% RSLogix 500 project DMINFEED - ONSITE - 17-01-07 - AFTER CHANGES.RSS, saved by version 7.00.00.19 %
PROJECT "DMINFEED"    % processor: SLC 500, 1747-L541 %

PROGRAM FILES
  LAD 2 "MAIN"  16 rungs
  LAD 3 "DECK1 TILT"  21 rungs
  LAD 4 "DECK2 TILT"  18 rungs
  LAD 5 "LUGLOADER"  18 rungs
  LAD 6 "SPARE"  1 rungs
  LAD 7 "DECK1 MOTS"  53 rungs
  LAD 8 "EXTRACTFAN"  7 rungs
  LAD 9 "BLOCKTX"  2 rungs
  LAD 14 "DECK2 MOTS"  23 rungs
  LAD 15 "ENCODER"  4 rungs
  LAD 16 "FEED_CONTR"  7 rungs
  LAD 17 "SCELUGLOAD"  11 rungs
  LAD 18 "REPORTING"  4 rungs
  LAD 20 "FILLET SYS"  28 rungs

DATA FILES
  O0 OUTPUT  39 elements
  I1 INPUT  46 elements
  S2 STATUS  164 elements
  B3 BINARY  100 elements
  T4 TIMER  100 elements
  C5 COUNTER  100 elements
  R6 CONTROL  1 elements
  N7 INTEGER  100 elements
  F8 FLOAT  1 elements
  N9 REMOTE IO  20 elements
  N10   100 elements
  N11 SCE SYSTEM  101 elements
  T12 SCE TIMER  11 elements
  N13   42 elements
  T14   30 elements
  C15   30 elements
  B16   100 elements

LADDER 2 "MAIN"
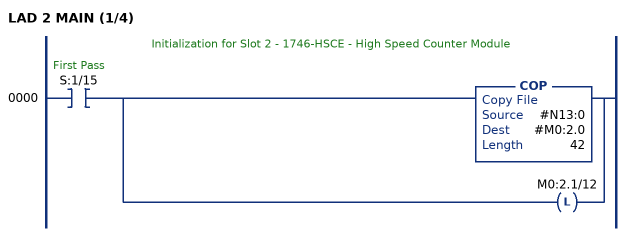
% Rung: 0 %
% Initialization for Slot 2 - 1746-HSCE - High Speed Counter Module %
SOR XIC S:1/15 BST COP #N13:0 #M0:2.0 42 NXB OTL M0:2.1/12 BND EOR
%   S:1/15  "First Pass" %

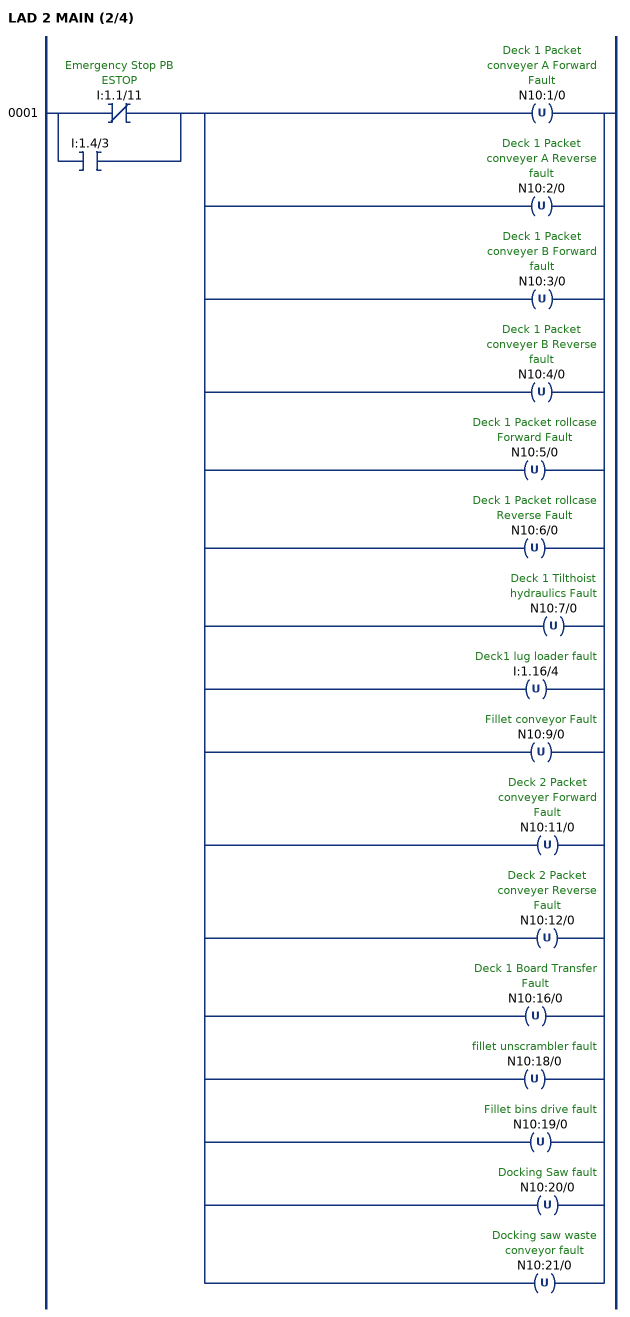
% Rung: 1 %
SOR BST XIO I:1.1/11 NXB XIC I:1.4/3 BND BST OTU N10:1/0 NXB OTU N10:2/0 NXB OTU N10:3/0 NXB OTU N10:4/0 NXB OTU N10:5/0 NXB OTU N10:6/0 NXB OTU N10:7/0 NXB OTU I:1.16/4 NXB OTU N10:9/0 NXB OTU N10:11/0 NXB OTU N10:12/0 NXB OTU N10:16/0 NXB OTU N10:18/0 NXB OTU N10:19/0 NXB OTU N10:20/0 NXB OTU N10:21/0 BND EOR
%   I:1.1/11  ESTOP  "Emergency Stop PB" %
%   N10:1/0  "Deck 1 Packet conveyer A Forward Fault" %
%   N10:2/0  "Deck 1 Packet conveyer A Reverse fault" %
%   N10:3/0  "Deck 1 Packet conveyer B Forward fault" %
%   N10:4/0  "Deck 1 Packet conveyer B Reverse fault" %
%   N10:5/0  "Deck 1 Packet rollcase Forward Fault" %
%   N10:6/0  "Deck 1 Packet rollcase Reverse Fault" %
%   N10:7/0  "Deck 1 Tilthoist hydraulics Fault" %
%   I:1.16/4  "Deck1 lug loader fault" %
%   N10:9/0  "Fillet conveyor Fault" %
%   N10:11/0  "Deck 2 Packet conveyer Forward Fault" %
%   N10:12/0  "Deck 2 Packet conveyer Reverse Fault" %
%   N10:16/0  "Deck 1 Board Transfer Fault" %
%   N10:18/0  "fillet unscrambler fault" %
%   N10:19/0  "Fillet bins drive fault" %
%   N10:20/0  "Docking Saw fault" %
%   N10:21/0  "Docking saw waste conveyor fault" %

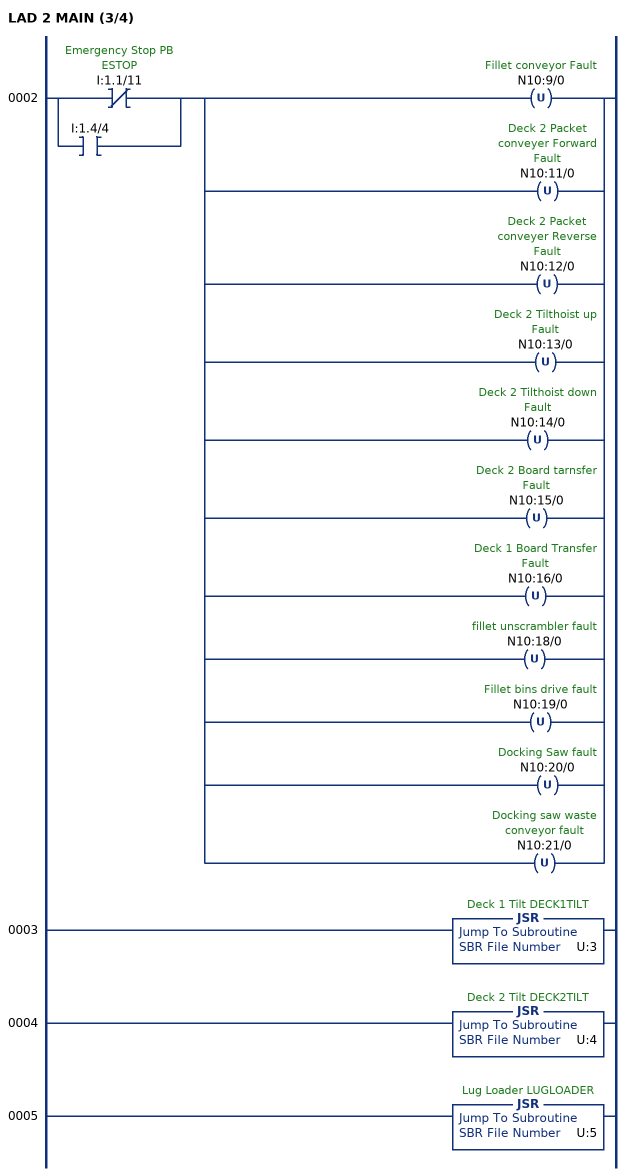
% Rung: 2 %
SOR BST XIO I:1.1/11 NXB XIC I:1.4/4 BND BST OTU N10:9/0 NXB OTU N10:11/0 NXB OTU N10:12/0 NXB OTU N10:13/0 NXB OTU N10:14/0 NXB OTU N10:15/0 NXB OTU N10:16/0 NXB OTU N10:18/0 NXB OTU N10:19/0 NXB OTU N10:20/0 NXB OTU N10:21/0 BND EOR
%   I:1.1/11  ESTOP  "Emergency Stop PB" %
%   N10:9/0  "Fillet conveyor Fault" %
%   N10:11/0  "Deck 2 Packet conveyer Forward Fault" %
%   N10:12/0  "Deck 2 Packet conveyer Reverse Fault" %
%   N10:13/0  "Deck 2 Tilthoist up Fault" %
%   N10:14/0  "Deck 2 Tilthoist down Fault" %
%   N10:15/0  "Deck 2 Board tarnsfer Fault" %
%   N10:16/0  "Deck 1 Board Transfer Fault" %
%   N10:18/0  "fillet unscrambler fault" %
%   N10:19/0  "Fillet bins drive fault" %
%   N10:20/0  "Docking Saw fault" %
%   N10:21/0  "Docking saw waste conveyor fault" %
% Rung: 3 %
SOR JSR U:3 EOR
%   U:3  DECK1TILT  "Deck 1 Tilt" %
% Rung: 4 %
SOR JSR U:4 EOR
%   U:4  DECK2TILT  "Deck 2 Tilt" %
% Rung: 5 %
SOR JSR U:5 EOR
%   U:5  LUGLOADER  "Lug Loader" %

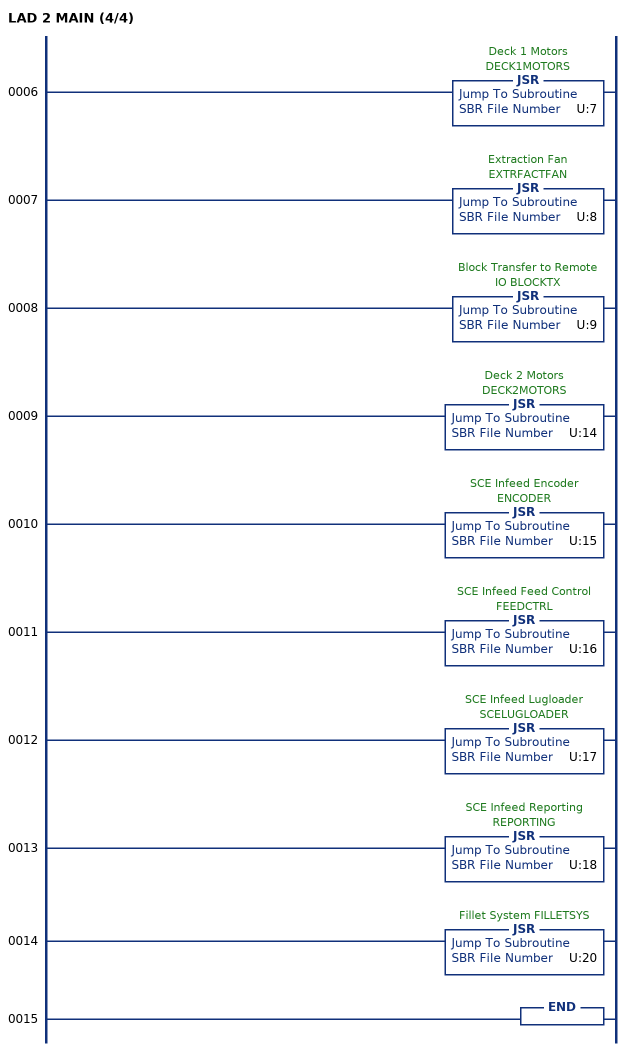
% Rung: 6 %
SOR JSR U:7 EOR
%   U:7  DECK1MOTORS  "Deck 1 Motors" %
% Rung: 7 %
SOR JSR U:8 EOR
%   U:8  EXTRFACTFAN  "Extraction Fan" %
% Rung: 8 %
SOR JSR U:9 EOR
%   U:9  BLOCKTX  "Block Transfer to Remote IO" %
% Rung: 9 %
SOR JSR U:14 EOR
%   U:14  DECK2MOTORS  "Deck 2 Motors" %
% Rung: 10 %
SOR JSR U:15 EOR
%   U:15  ENCODER  "SCE Infeed Encoder" %
% Rung: 11 %
SOR JSR U:16 EOR
%   U:16  FEEDCTRL  "SCE Infeed Feed Control" %
% Rung: 12 %
SOR JSR U:17 EOR
%   U:17  SCELUGLOADER  "SCE Infeed Lugloader" %
% Rung: 13 %
SOR JSR U:18 EOR
%   U:18  REPORTING  "SCE Infeed Reporting" %
% Rung: 14 %
SOR JSR U:20 EOR
%   U:20  FILLETSYS  "Fillet System" %
% Rung: 15 %
SOR END EOR

LADDER 3 "DECK1 TILT"
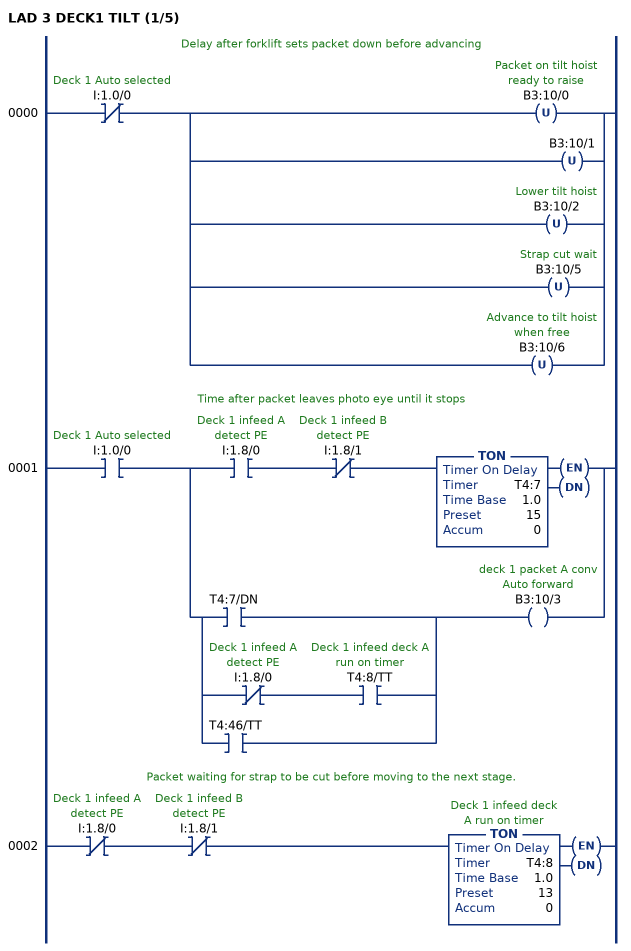
% Rung: 0 %
% Delay after forklift sets packet down before advancing %
SOR XIO I:1.0/0 BST OTU B3:10/0 NXB OTU B3:10/1 NXB OTU B3:10/2 NXB OTU B3:10/5 NXB OTU B3:10/6 BND EOR
%   I:1.0/0  "Deck 1 Auto selected" %
%   B3:10/0  "Packet on tilt hoist ready to raise" %
%   B3:10/2  "Lower tilt hoist" %
%   B3:10/5  "Strap cut wait" %
%   B3:10/6  "Advance to tilt hoist when free" %
% Rung: 1 %
% Time after packet leaves photo eye until it stops %
SOR XIC I:1.0/0 BST XIC I:1.8/0 XIO I:1.8/1 TON T4:7 1.0 15 0 NXB BST XIC T4:7/DN NXB XIO I:1.8/0 XIC T4:8/TT NXB XIC T4:46/TT BND OTE B3:10/3 BND EOR
%   I:1.0/0  "Deck 1 Auto selected" %
%   I:1.8/0  "Deck 1 infeed A detect PE" %
%   I:1.8/1  "Deck 1 infeed B detect PE" %
%   T4:8  "Deck 1 infeed deck A run on timer" %
%   B3:10/3  "deck 1 packet A conv Auto forward" %
% Rung: 2 %
% Packet waiting for strap to be cut before moving to the next stage. %
SOR XIO I:1.8/0 XIO I:1.8/1 TON T4:8 1.0 13 0 EOR
%   I:1.8/0  "Deck 1 infeed A detect PE" %
%   I:1.8/1  "Deck 1 infeed B detect PE" %
%   T4:8  "Deck 1 infeed deck A run on timer" %

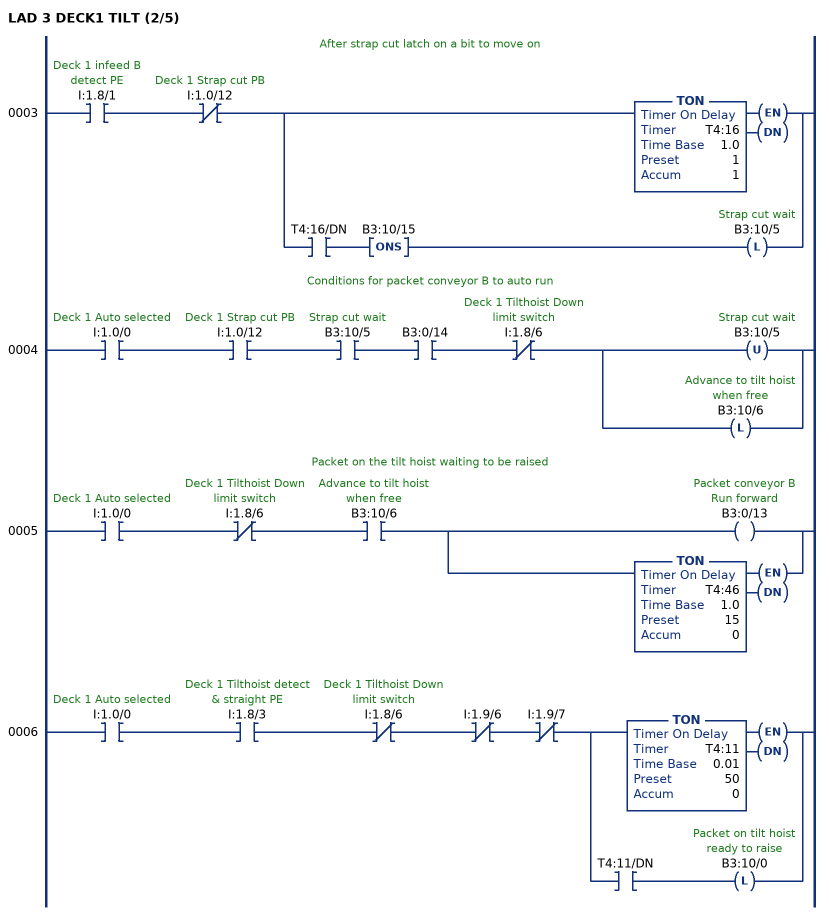
% Rung: 3 %
% After strap cut latch on a bit to move on %
SOR XIC I:1.8/1 XIO I:1.0/12 BST TON T4:16 1.0 1 1 NXB XIC T4:16/DN OSR B3:10/15 OTL B3:10/5 BND EOR
%   I:1.8/1  "Deck 1 infeed B detect PE" %
%   I:1.0/12  "Deck 1 Strap cut PB" %
%   B3:10/5  "Strap cut wait" %
% Rung: 4 %
% Conditions for packet conveyor B to auto run %
SOR XIC I:1.0/0 XIC I:1.0/12 XIC B3:10/5 XIC B3:0/14 XIO I:1.8/6 BST OTU B3:10/5 NXB OTL B3:10/6 BND EOR
%   I:1.0/0  "Deck 1 Auto selected" %
%   I:1.0/12  "Deck 1 Strap cut PB" %
%   B3:10/5  "Strap cut wait" %
%   I:1.8/6  "Deck 1 Tilthoist Down limit switch" %
%   B3:10/6  "Advance to tilt hoist when free" %
% Rung: 5 %
% Packet on the tilt hoist waiting to be raised %
SOR XIC I:1.0/0 XIO I:1.8/6 XIC B3:10/6 BST OTE B3:0/13 NXB TON T4:46 1.0 15 0 BND EOR
%   I:1.0/0  "Deck 1 Auto selected" %
%   I:1.8/6  "Deck 1 Tilthoist Down limit switch" %
%   B3:10/6  "Advance to tilt hoist when free" %
%   B3:0/13  "Packet conveyor B Run forward" %
% Rung: 6 %
SOR XIC I:1.0/0 XIC I:1.8/3 XIO I:1.8/6 XIO I:1.9/6 XIO I:1.9/7 BST TON T4:11 0.01 50 0 NXB XIC T4:11/DN OTL B3:10/0 BND EOR
%   I:1.0/0  "Deck 1 Auto selected" %
%   I:1.8/3  "Deck 1 Tilthoist detect & straight PE" %
%   I:1.8/6  "Deck 1 Tilthoist Down limit switch" %
%   B3:10/0  "Packet on tilt hoist ready to raise" %

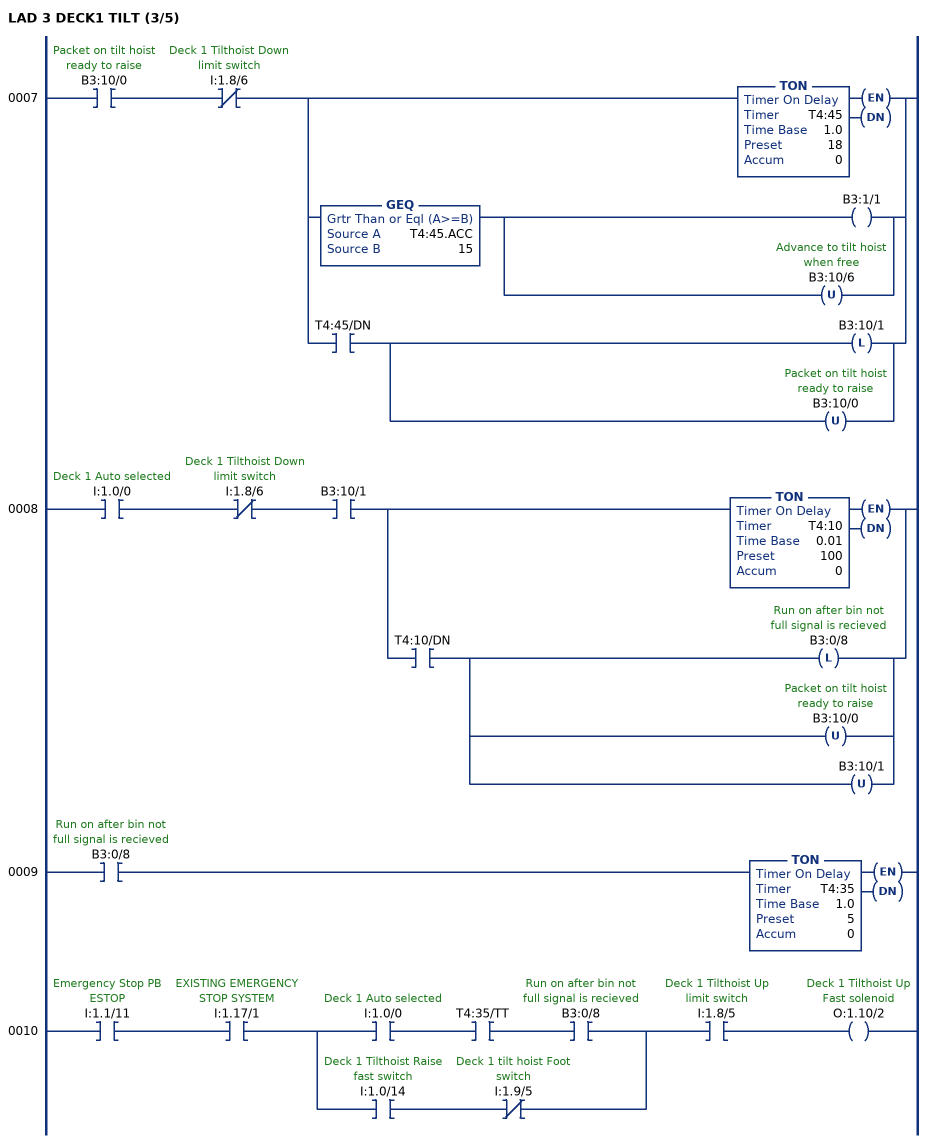
% Rung: 7 %
SOR XIC B3:10/0 XIO I:1.8/6 BST TON T4:45 1.0 18 0 NXB GEQ T4:45.ACC 15 BST OTE B3:1/1 NXB OTU B3:10/6 BND NXB XIC T4:45/DN BST OTL B3:10/1 NXB OTU B3:10/0 BND BND EOR
%   B3:10/0  "Packet on tilt hoist ready to raise" %
%   I:1.8/6  "Deck 1 Tilthoist Down limit switch" %
%   B3:10/6  "Advance to tilt hoist when free" %
% Rung: 8 %
SOR XIC I:1.0/0 XIO I:1.8/6 XIC B3:10/1 BST TON T4:10 0.01 100 0 NXB XIC T4:10/DN BST OTL B3:0/8 NXB OTU B3:10/0 NXB OTU B3:10/1 BND BND EOR
%   I:1.0/0  "Deck 1 Auto selected" %
%   I:1.8/6  "Deck 1 Tilthoist Down limit switch" %
%   B3:0/8  "Run on after bin not full signal is recieved" %
%   B3:10/0  "Packet on tilt hoist ready to raise" %
% Rung: 9 %
SOR XIC B3:0/8 TON T4:35 1.0 5 0 EOR
%   B3:0/8  "Run on after bin not full signal is recieved" %
% Rung: 10 %
SOR XIC I:1.1/11 XIC I:1.17/1 BST XIC I:1.0/0 XIC T4:35/TT XIC B3:0/8 NXB XIC I:1.0/14 XIO I:1.9/5 BND XIC I:1.8/5 OTE O:1.10/2 EOR
%   I:1.1/11  ESTOP  "Emergency Stop PB" %
%   I:1.17/1  "EXISTING EMERGENCY STOP SYSTEM" %
%   I:1.0/0  "Deck 1 Auto selected" %
%   B3:0/8  "Run on after bin not full signal is recieved" %
%   I:1.0/14  "Deck 1 Tilthoist Raise fast switch" %
%   I:1.9/5  "Deck 1 tilt hoist Foot switch" %
%   I:1.8/5  "Deck 1 Tilthoist Up limit switch" %
%   O:1.10/2  "Deck 1 Tilthoist Up Fast solenoid" %

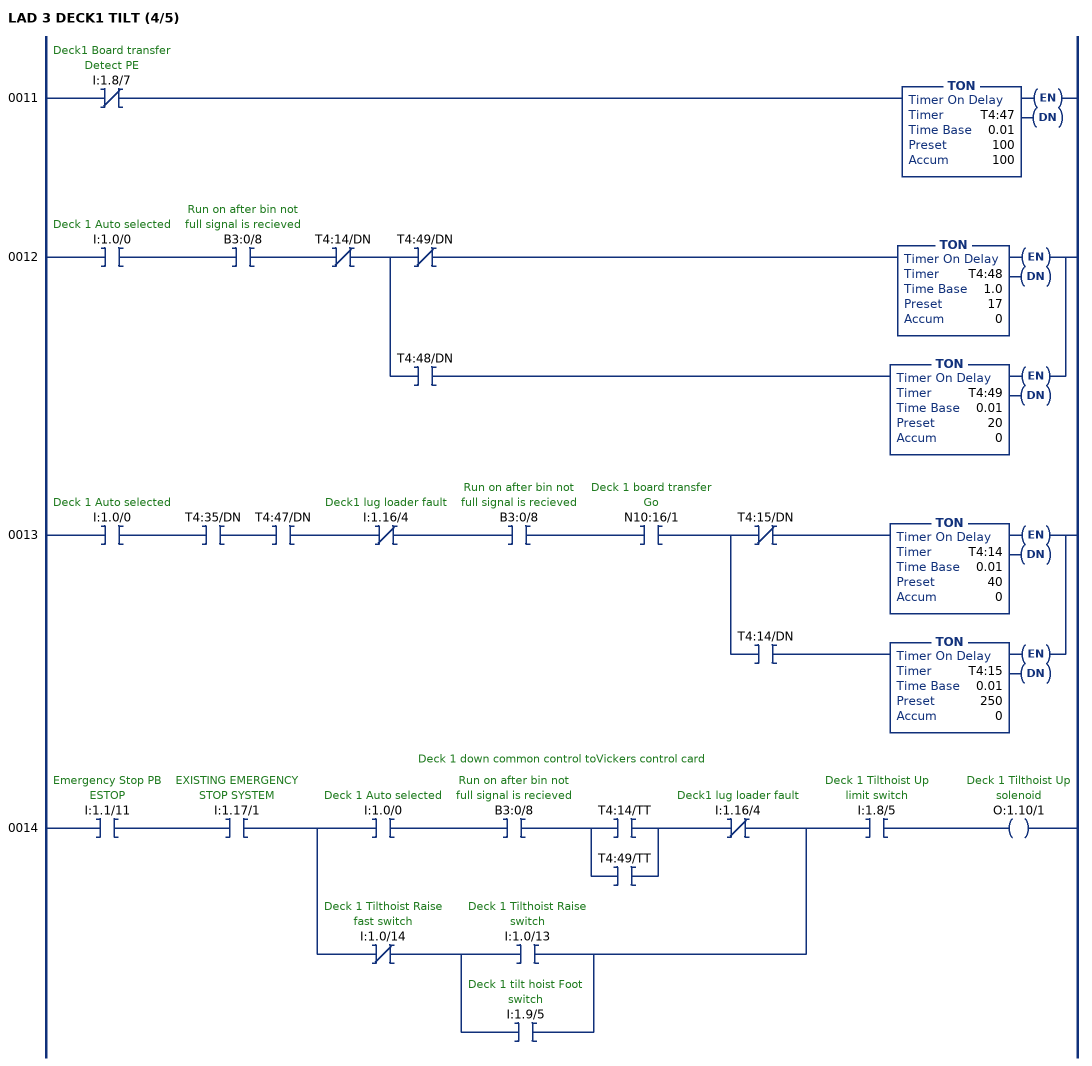
% Rung: 11 %
SOR XIO I:1.8/7 TON T4:47 0.01 100 100 EOR
%   I:1.8/7  "Deck1 Board transfer Detect PE" %
% Rung: 12 %
SOR XIC I:1.0/0 XIC B3:0/8 XIO T4:14/DN BST XIO T4:49/DN TON T4:48 1.0 17 0 NXB XIC T4:48/DN TON T4:49 0.01 20 0 BND EOR
%   I:1.0/0  "Deck 1 Auto selected" %
%   B3:0/8  "Run on after bin not full signal is recieved" %
% Rung: 13 %
SOR XIC I:1.0/0 XIC T4:35/DN XIC T4:47/DN XIO I:1.16/4 XIC B3:0/8 XIC N10:16/1 BST XIO T4:15/DN TON T4:14 0.01 40 0 NXB XIC T4:14/DN TON T4:15 0.01 250 0 BND EOR
%   I:1.0/0  "Deck 1 Auto selected" %
%   I:1.16/4  "Deck1 lug loader fault" %
%   B3:0/8  "Run on after bin not full signal is recieved" %
%   N10:16/1  "Deck 1 board transfer Go" %
% Rung: 14 %
% Deck 1 down common control toVickers control card %
SOR XIC I:1.1/11 XIC I:1.17/1 BST XIC I:1.0/0 XIC B3:0/8 BST XIC T4:14/TT NXB XIC T4:49/TT BND XIO I:1.16/4 NXB XIO I:1.0/14 BST XIC I:1.0/13 NXB XIC I:1.9/5 BND BND XIC I:1.8/5 OTE O:1.10/1 EOR
%   I:1.1/11  ESTOP  "Emergency Stop PB" %
%   I:1.17/1  "EXISTING EMERGENCY STOP SYSTEM" %
%   I:1.0/0  "Deck 1 Auto selected" %
%   B3:0/8  "Run on after bin not full signal is recieved" %
%   I:1.16/4  "Deck1 lug loader fault" %
%   I:1.0/14  "Deck 1 Tilthoist Raise fast switch" %
%   I:1.0/13  "Deck 1 Tilthoist Raise switch" %
%   I:1.9/5  "Deck 1 tilt hoist Foot switch" %
%   I:1.8/5  "Deck 1 Tilthoist Up limit switch" %
%   O:1.10/1  "Deck 1 Tilthoist Up solenoid" %

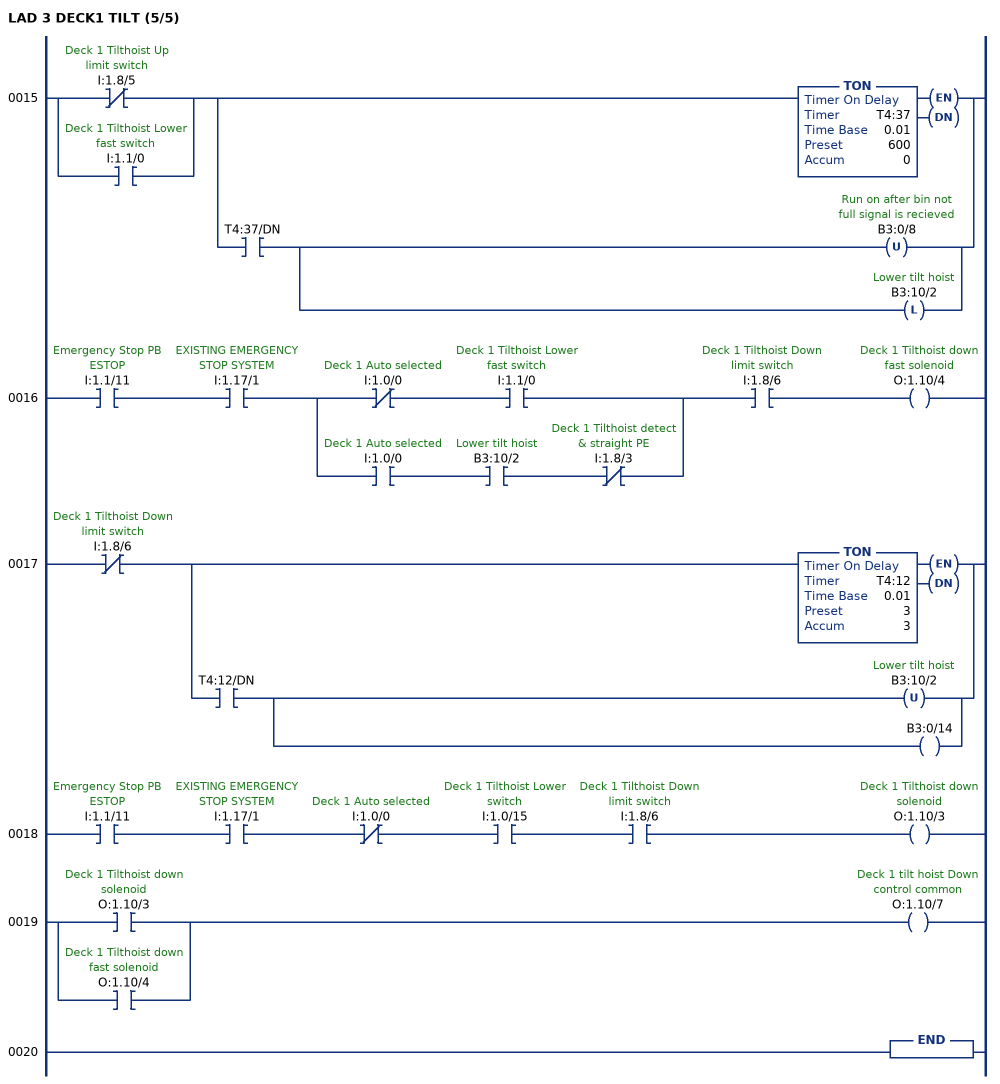
% Rung: 15 %
SOR BST XIO I:1.8/5 NXB XIC I:1.1/0 BND BST TON T4:37 0.01 600 0 NXB XIC T4:37/DN BST OTU B3:0/8 NXB OTL B3:10/2 BND BND EOR
%   I:1.8/5  "Deck 1 Tilthoist Up limit switch" %
%   I:1.1/0  "Deck 1 Tilthoist Lower fast switch" %
%   B3:0/8  "Run on after bin not full signal is recieved" %
%   B3:10/2  "Lower tilt hoist" %
% Rung: 16 %
SOR XIC I:1.1/11 XIC I:1.17/1 BST XIO I:1.0/0 XIC I:1.1/0 NXB XIC I:1.0/0 XIC B3:10/2 XIO I:1.8/3 BND XIC I:1.8/6 OTE O:1.10/4 EOR
%   I:1.1/11  ESTOP  "Emergency Stop PB" %
%   I:1.17/1  "EXISTING EMERGENCY STOP SYSTEM" %
%   I:1.0/0  "Deck 1 Auto selected" %
%   I:1.1/0  "Deck 1 Tilthoist Lower fast switch" %
%   B3:10/2  "Lower tilt hoist" %
%   I:1.8/3  "Deck 1 Tilthoist detect & straight PE" %
%   I:1.8/6  "Deck 1 Tilthoist Down limit switch" %
%   O:1.10/4  "Deck 1 Tilthoist down fast solenoid" %
% Rung: 17 %
SOR XIO I:1.8/6 BST TON T4:12 0.01 3 3 NXB XIC T4:12/DN BST OTU B3:10/2 NXB OTE B3:0/14 BND BND EOR
%   I:1.8/6  "Deck 1 Tilthoist Down limit switch" %
%   B3:10/2  "Lower tilt hoist" %
% Rung: 18 %
SOR XIC I:1.1/11 XIC I:1.17/1 XIO I:1.0/0 XIC I:1.0/15 XIC I:1.8/6 OTE O:1.10/3 EOR
%   I:1.1/11  ESTOP  "Emergency Stop PB" %
%   I:1.17/1  "EXISTING EMERGENCY STOP SYSTEM" %
%   I:1.0/0  "Deck 1 Auto selected" %
%   I:1.0/15  "Deck 1 Tilthoist Lower switch" %
%   I:1.8/6  "Deck 1 Tilthoist Down limit switch" %
%   O:1.10/3  "Deck 1 Tilthoist down solenoid" %
% Rung: 19 %
SOR BST XIC O:1.10/3 NXB XIC O:1.10/4 BND OTE O:1.10/7 EOR
%   O:1.10/3  "Deck 1 Tilthoist down solenoid" %
%   O:1.10/4  "Deck 1 Tilthoist down fast solenoid" %
%   O:1.10/7  "Deck 1 tilt hoist Down control common" %
% Rung: 20 %
SOR END EOR

LADDER 4 "DECK2 TILT"
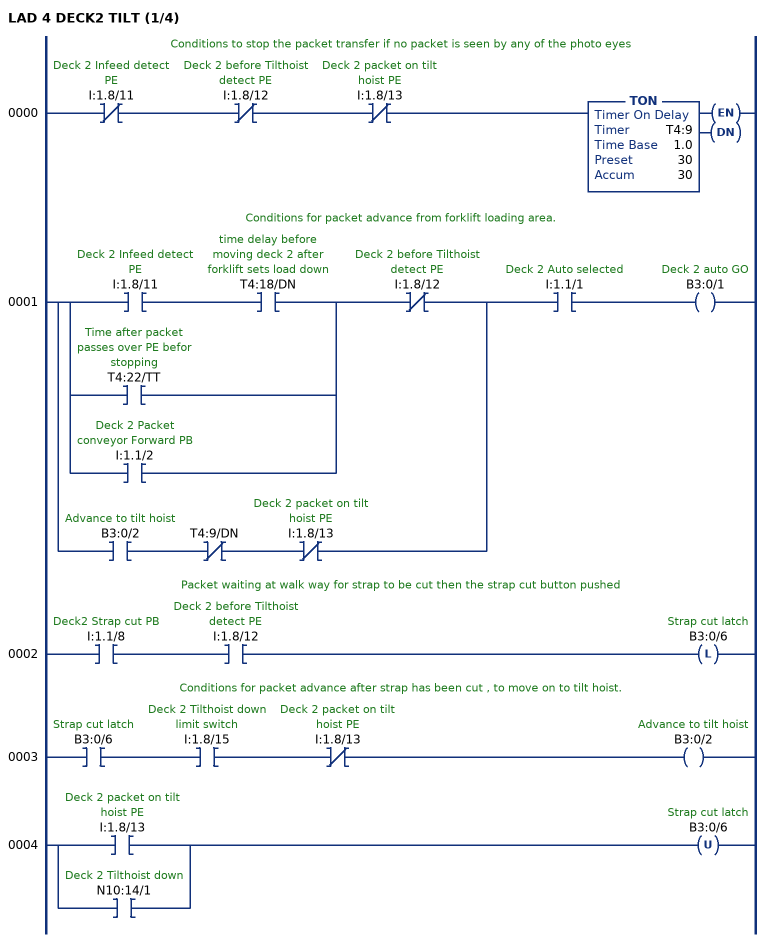
% Rung: 0 %
% Conditions to stop the packet transfer if no packet is seen by any of the photo eyes %
SOR XIO I:1.8/11 XIO I:1.8/12 XIO I:1.8/13 TON T4:9 1.0 30 30 EOR
%   I:1.8/11  "Deck 2 Infeed detect PE" %
%   I:1.8/12  "Deck 2 before Tilthoist detect PE" %
%   I:1.8/13  "Deck 2 packet on tilt hoist PE" %
% Rung: 1 %
% Conditions for packet advance from forklift loading area. %
SOR BST BST XIC I:1.8/11 XIC T4:18/DN NXB BST XIC T4:22/TT NXB XIC I:1.1/2 BND BND XIO I:1.8/12 NXB XIC B3:0/2 XIO T4:9/DN XIO I:1.8/13 BND XIC I:1.1/1 OTE B3:0/1 EOR
%   I:1.8/11  "Deck 2 Infeed detect PE" %
%   T4:18  "time delay before moving deck 2 after forklift sets load down" %
%   T4:22  "Time after packet passes over PE befor stopping" %
%   I:1.1/2  "Deck 2 Packet conveyor Forward PB" %
%   I:1.8/12  "Deck 2 before Tilthoist detect PE" %
%   B3:0/2  "Advance to tilt hoist" %
%   I:1.8/13  "Deck 2 packet on tilt hoist PE" %
%   I:1.1/1  "Deck 2 Auto selected" %
%   B3:0/1  "Deck 2 auto GO" %
% Rung: 2 %
% Packet waiting at walk way for strap to be cut then the strap cut button pushed %
SOR XIC I:1.1/8 XIC I:1.8/12 OTL B3:0/6 EOR
%   I:1.1/8  "Deck2 Strap cut PB" %
%   I:1.8/12  "Deck 2 before Tilthoist detect PE" %
%   B3:0/6  "Strap cut latch" %
% Rung: 3 %
% Conditions for packet advance after strap has been cut , to move on to tilt hoist. %
SOR XIC B3:0/6 XIC I:1.8/15 XIO I:1.8/13 OTE B3:0/2 EOR
%   B3:0/6  "Strap cut latch" %
%   I:1.8/15  "Deck 2 Tilthoist down limit switch" %
%   I:1.8/13  "Deck 2 packet on tilt hoist PE" %
%   B3:0/2  "Advance to tilt hoist" %
% Rung: 4 %
SOR BST XIC I:1.8/13 NXB XIC N10:14/1 BND OTU B3:0/6 EOR
%   I:1.8/13  "Deck 2 packet on tilt hoist PE" %
%   N10:14/1  "Deck 2 Tilthoist down" %
%   B3:0/6  "Strap cut latch" %

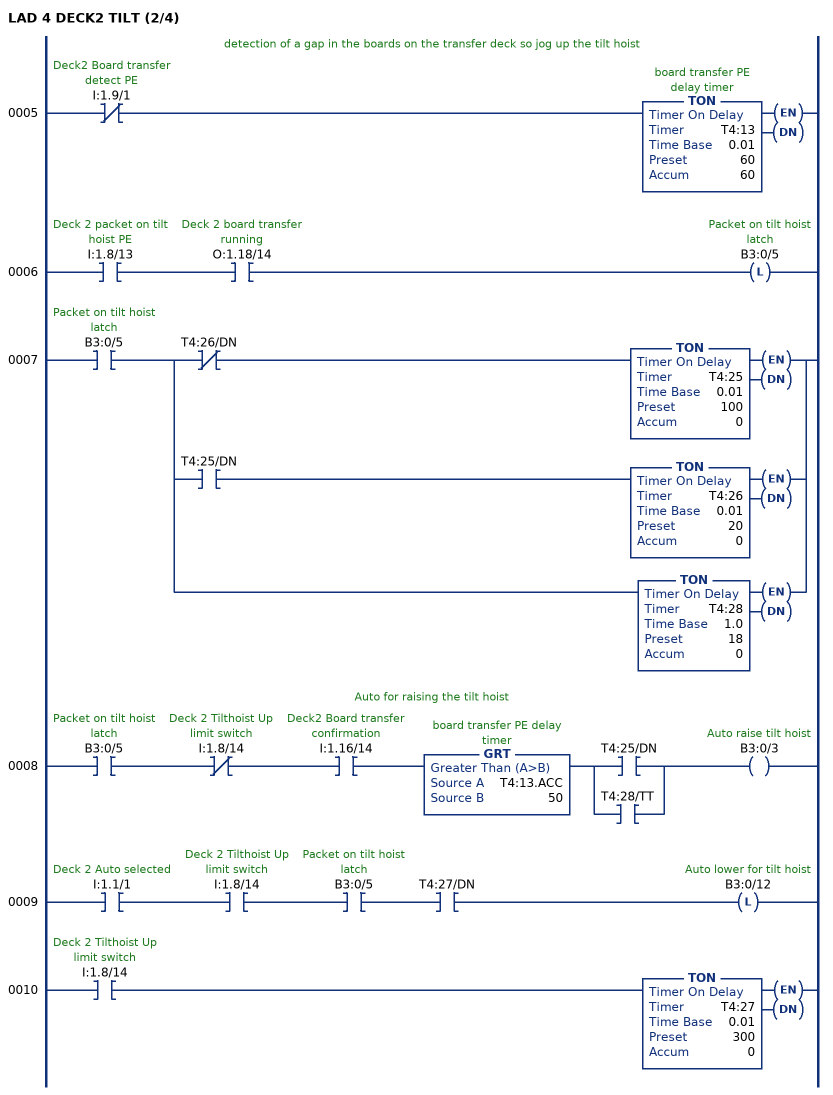
% Rung: 5 %
% detection of a gap in the boards on the transfer deck so jog up the tilt hoist %
SOR XIO I:1.9/1 TON T4:13 0.01 60 60 EOR
%   I:1.9/1  "Deck2 Board transfer detect PE" %
%   T4:13  "board transfer PE delay timer" %
% Rung: 6 %
SOR XIC I:1.8/13 XIC O:1.18/14 OTL B3:0/5 EOR
%   I:1.8/13  "Deck 2 packet on tilt hoist PE" %
%   O:1.18/14  "Deck 2 board transfer running" %
%   B3:0/5  "Packet on tilt hoist latch" %
% Rung: 7 %
SOR XIC B3:0/5 BST XIO T4:26/DN TON T4:25 0.01 100 0 NXB BST XIC T4:25/DN TON T4:26 0.01 20 0 NXB TON T4:28 1.0 18 0 BND BND EOR
%   B3:0/5  "Packet on tilt hoist latch" %
% Rung: 8 %
% Auto for raising the tilt hoist %
SOR XIC B3:0/5 XIO I:1.8/14 XIC I:1.16/14 GRT T4:13.ACC 50 BST XIC T4:25/DN NXB XIC T4:28/TT BND OTE B3:0/3 EOR
%   B3:0/5  "Packet on tilt hoist latch" %
%   I:1.8/14  "Deck 2 Tilthoist Up limit switch" %
%   I:1.16/14  "Deck2 Board transfer confirmation" %
%   T4:13  "board transfer PE delay timer" %
%   B3:0/3  "Auto raise tilt hoist" %
% Rung: 9 %
SOR XIC I:1.1/1 XIC I:1.8/14 XIC B3:0/5 XIC T4:27/DN OTL B3:0/12 EOR
%   I:1.1/1  "Deck 2 Auto selected" %
%   I:1.8/14  "Deck 2 Tilthoist Up limit switch" %
%   B3:0/5  "Packet on tilt hoist latch" %
%   B3:0/12  "Auto lower for tilt hoist" %
% Rung: 10 %
SOR XIC I:1.8/14 TON T4:27 0.01 300 0 EOR
%   I:1.8/14  "Deck 2 Tilthoist Up limit switch" %

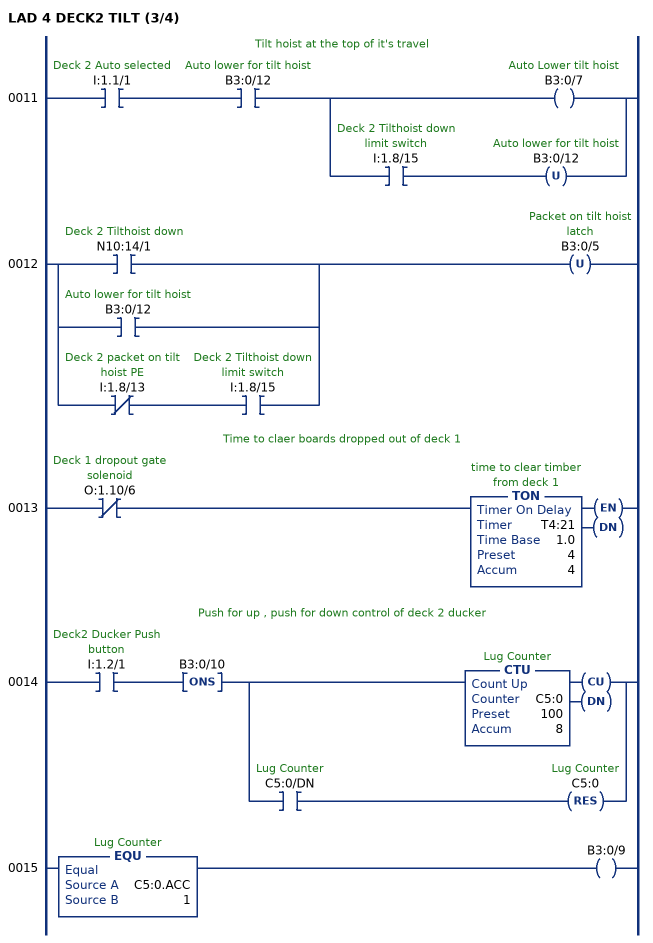
% Rung: 11 %
% Tilt hoist at the top of it's travel %
SOR XIC I:1.1/1 XIC B3:0/12 BST OTE B3:0/7 NXB XIC I:1.8/15 OTU B3:0/12 BND EOR
%   I:1.1/1  "Deck 2 Auto selected" %
%   B3:0/12  "Auto lower for tilt hoist" %
%   B3:0/7  "Auto Lower tilt hoist" %
%   I:1.8/15  "Deck 2 Tilthoist down limit switch" %
% Rung: 12 %
SOR BST BST XIC N10:14/1 NXB XIC B3:0/12 BND NXB XIO I:1.8/13 XIC I:1.8/15 BND OTU B3:0/5 EOR
%   N10:14/1  "Deck 2 Tilthoist down" %
%   B3:0/12  "Auto lower for tilt hoist" %
%   I:1.8/13  "Deck 2 packet on tilt hoist PE" %
%   I:1.8/15  "Deck 2 Tilthoist down limit switch" %
%   B3:0/5  "Packet on tilt hoist latch" %
% Rung: 13 %
% Time to claer boards dropped out of deck 1 %
SOR XIO O:1.10/6 TON T4:21 1.0 4 4 EOR
%   O:1.10/6  "Deck 1 dropout gate solenoid" %
%   T4:21  "time to clear timber from deck 1" %
% Rung: 14 %
% Push for up , push for down control of deck 2 ducker %
SOR XIC I:1.2/1 OSR B3:0/10 BST CTU C5:0 100 8 NXB XIC C5:0/DN RES C5:0 BND EOR
%   I:1.2/1  "Deck2 Ducker Push button" %
%   C5:0  "Lug Counter" %
% Rung: 15 %
SOR EQU C5:0.ACC 1 OTE B3:0/9 EOR
%   C5:0  "Lug Counter" %

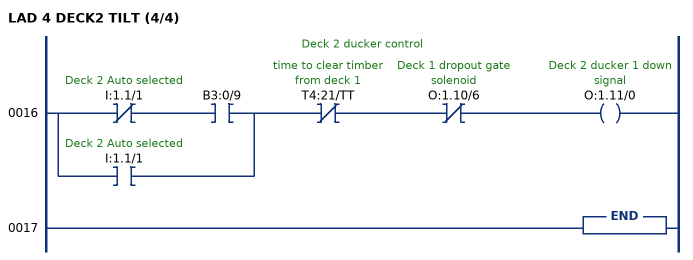
% Rung: 16 %
% Deck 2 ducker control %
SOR BST XIO I:1.1/1 XIC B3:0/9 NXB XIC I:1.1/1 BND XIO T4:21/TT XIO O:1.10/6 OTE O:1.11/0 EOR
%   I:1.1/1  "Deck 2 Auto selected" %
%   T4:21  "time to clear timber from deck 1" %
%   O:1.10/6  "Deck 1 dropout gate solenoid" %
%   O:1.11/0  "Deck 2 ducker 1 down signal" %
% Rung: 17 %
SOR END EOR

LADDER 5 "LUGLOADER"
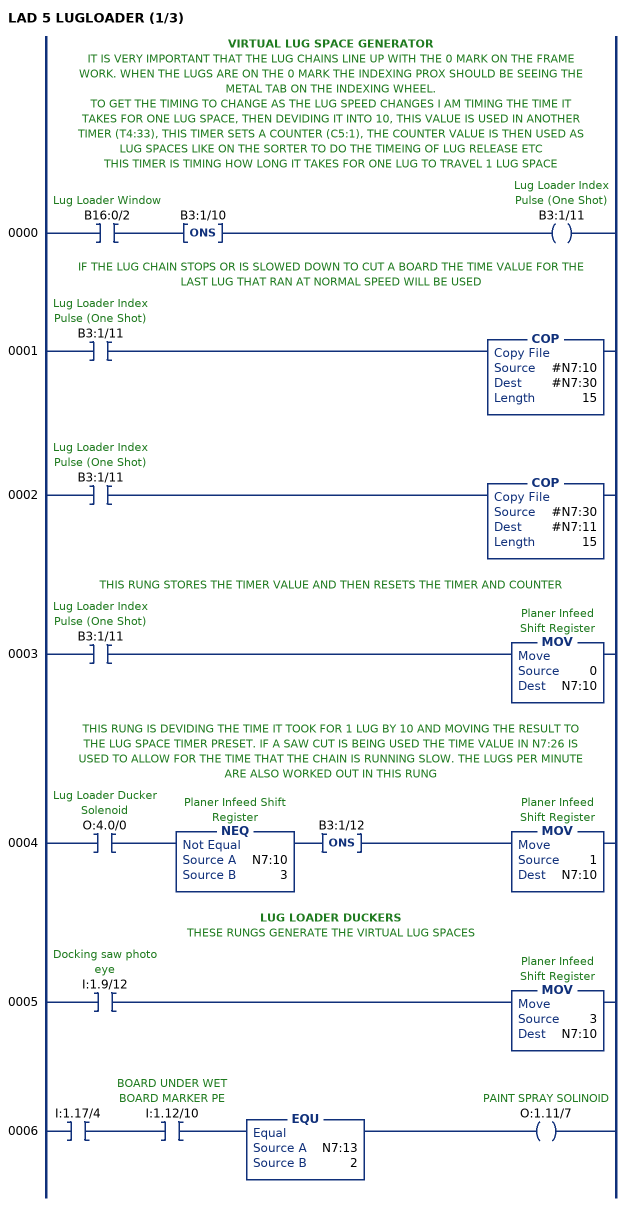
% Rung: 0 %
% TITLE: VIRTUAL LUG SPACE GENERATOR %
% IT IS VERY IMPORTANT THAT THE LUG CHAINS LINE UP WITH THE 0 MARK ON THE FRAME WORK. WHEN THE LUGS ARE ON THE 0 MARK THE INDEXING PROX SHOULD BE SEEING THE METAL TAB ON THE INDEXING WHEEL.
% TO GET THE TIMING TO CHANGE AS THE LUG SPEED CHANGES I AM TIMING THE TIME IT TAKES FOR ONE LUG SPACE, THEN DEVIDING IT INTO 10, THIS VALUE IS USED IN ANOTHER TIMER (T4:33), THIS TIMER SETS A COUNTER (C5:1), THE COUNTER VALUE IS THEN USED AS LUG SPACES LIKE ON THE SORTER TO DO THE TIMEING OF LUG RELEASE ETC
% THIS TIMER IS TIMING HOW LONG IT TAKES FOR ONE LUG TO TRAVEL 1 LUG SPACE %
SOR XIC B16:0/2 OSR B3:1/10 OTE B3:1/11 EOR
%   B16:0/2  "Lug Loader Window" %
%   B3:1/11  "Lug Loader Index Pulse (One Shot)" %
% Rung: 1 %
% IF THE LUG CHAIN STOPS OR IS SLOWED DOWN TO CUT A BOARD THE TIME VALUE FOR THE LAST LUG THAT RAN AT NORMAL SPEED WILL BE USED %
SOR XIC B3:1/11 COP #N7:10 #N7:30 15 EOR
%   B3:1/11  "Lug Loader Index Pulse (One Shot)" %
%   N7:10  "Planer Infeed Shift Register" %
% Rung: 2 %
SOR XIC B3:1/11 COP #N7:30 #N7:11 15 EOR
%   B3:1/11  "Lug Loader Index Pulse (One Shot)" %
% Rung: 3 %
% THIS RUNG STORES THE TIMER VALUE AND THEN RESETS THE TIMER AND COUNTER %
SOR XIC B3:1/11 MOV 0 N7:10 EOR
%   B3:1/11  "Lug Loader Index Pulse (One Shot)" %
%   N7:10  "Planer Infeed Shift Register" %
% Rung: 4 %
% THIS RUNG IS DEVIDING THE TIME IT TOOK FOR 1 LUG BY 10 AND MOVING THE RESULT TO THE LUG SPACE TIMER PRESET. IF A SAW CUT IS BEING USED THE TIME VALUE IN N7:26 IS USED TO ALLOW FOR THE TIME THAT THE CHAIN IS RUNNING SLOW. THE LUGS PER MINUTE ARE ALSO WORKED OUT IN THIS RUNG %
SOR XIC O:4.0/0 NEQ N7:10 3 OSR B3:1/12 MOV 1 N7:10 EOR
%   O:4.0/0  "Lug Loader Ducker Solenoid" %
%   N7:10  "Planer Infeed Shift Register" %
% Rung: 5 %
% TITLE: LUG LOADER DUCKERS %
% THESE RUNGS GENERATE THE VIRTUAL LUG SPACES %
SOR XIC I:1.9/12 MOV 3 N7:10 EOR
%   I:1.9/12  "Docking saw photo eye" %
%   N7:10  "Planer Infeed Shift Register" %
% Rung: 6 %
SOR XIC I:1.17/4 XIC I:1.12/10 EQU N7:13 2 OTE O:1.11/7 EOR
%   I:1.12/10  "BOARD UNDER WET BOARD MARKER PE" %
%   O:1.11/7  "PAINT SPRAY SOLINOID" %

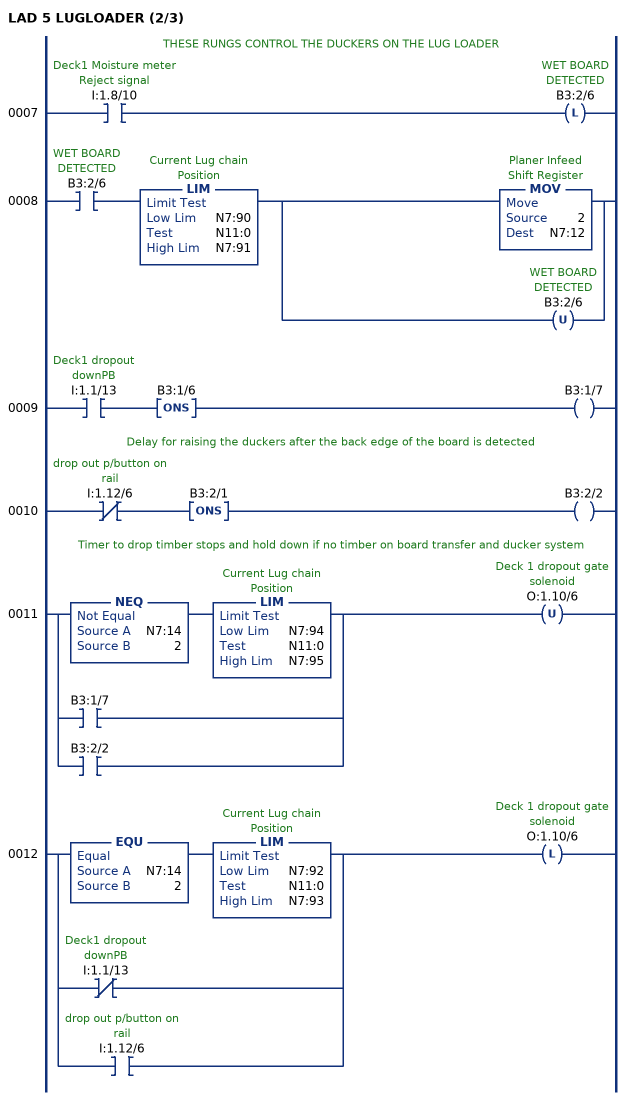
% Rung: 7 %
% THESE RUNGS CONTROL THE DUCKERS ON THE LUG LOADER %
SOR XIC I:1.8/10 OTL B3:2/6 EOR
%   I:1.8/10  "Deck1 Moisture meter Reject signal" %
%   B3:2/6  "WET BOARD DETECTED" %
% Rung: 8 %
SOR XIC B3:2/6 LIM N7:90 N11:0 N7:91 BST MOV 2 N7:12 NXB OTU B3:2/6 BND EOR
%   B3:2/6  "WET BOARD DETECTED" %
%   N11:0  "Current Lug chain Position" %
%   N7:12  "Planer Infeed Shift Register" %
% Rung: 9 %
SOR XIC I:1.1/13 OSR B3:1/6 OTE B3:1/7 EOR
%   I:1.1/13  "Deck1 dropout downPB" %
% Rung: 10 %
% Delay for raising the duckers after the back edge of the board is detected %
SOR XIO I:1.12/6 OSR B3:2/1 OTE B3:2/2 EOR
%   I:1.12/6  "drop out p/button on rail" %
% Rung: 11 %
% Timer to drop timber stops and hold down if no timber on board transfer and ducker system %
SOR BST NEQ N7:14 2 LIM N7:94 N11:0 N7:95 NXB XIC B3:1/7 NXB XIC B3:2/2 BND OTU O:1.10/6 EOR
%   N11:0  "Current Lug chain Position" %
%   O:1.10/6  "Deck 1 dropout gate solenoid" %
% Rung: 12 %
SOR BST EQU N7:14 2 LIM N7:92 N11:0 N7:93 NXB XIO I:1.1/13 NXB XIC I:1.12/6 BND OTL O:1.10/6 EOR
%   N11:0  "Current Lug chain Position" %
%   I:1.1/13  "Deck1 dropout downPB" %
%   I:1.12/6  "drop out p/button on rail" %
%   O:1.10/6  "Deck 1 dropout gate solenoid" %

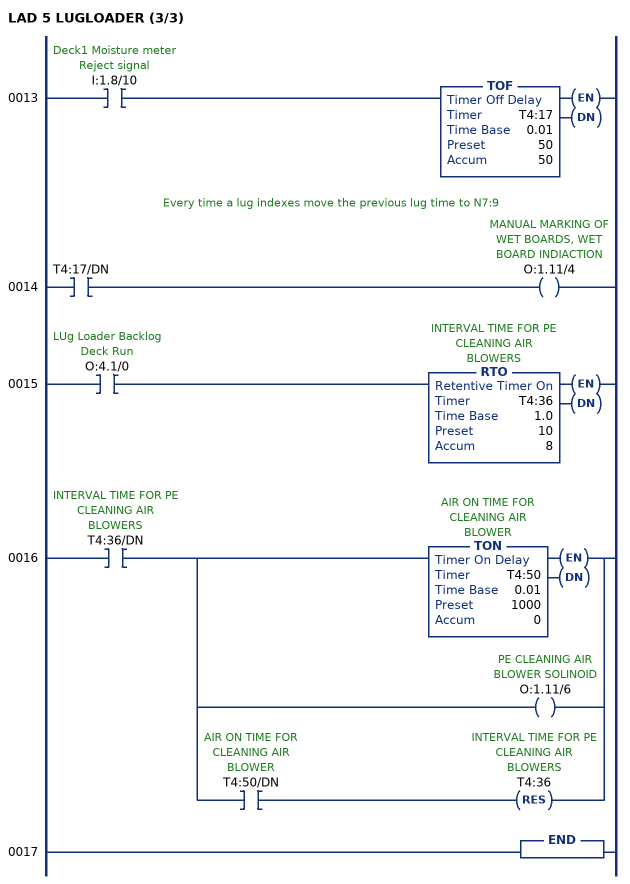
% Rung: 13 %
SOR XIC I:1.8/10 TOF T4:17 0.01 50 50 EOR
%   I:1.8/10  "Deck1 Moisture meter Reject signal" %
% Rung: 14 %
% Every time a lug indexes move the previous lug time to N7:9 %
SOR XIC T4:17/DN OTE O:1.11/4 EOR
%   O:1.11/4  "MANUAL MARKING OF WET BOARDS, WET BOARD INDIACTION" %
% Rung: 15 %
SOR XIC O:4.1/0 RTO T4:36 1.0 10 8 EOR
%   O:4.1/0  "LUg Loader Backlog Deck Run" %
%   T4:36  "INTERVAL TIME FOR PE CLEANING AIR BLOWERS" %
% Rung: 16 %
SOR XIC T4:36/DN BST TON T4:50 0.01 1000 0 NXB OTE O:1.11/6 NXB XIC T4:50/DN RES T4:36 BND EOR
%   T4:36  "INTERVAL TIME FOR PE CLEANING AIR BLOWERS" %
%   T4:50  "AIR ON TIME FOR CLEANING AIR BLOWER" %
%   O:1.11/6  "PE CLEANING AIR BLOWER SOLINOID" %
% Rung: 17 %
SOR END EOR

LADDER 7 "DECK1 MOTS"
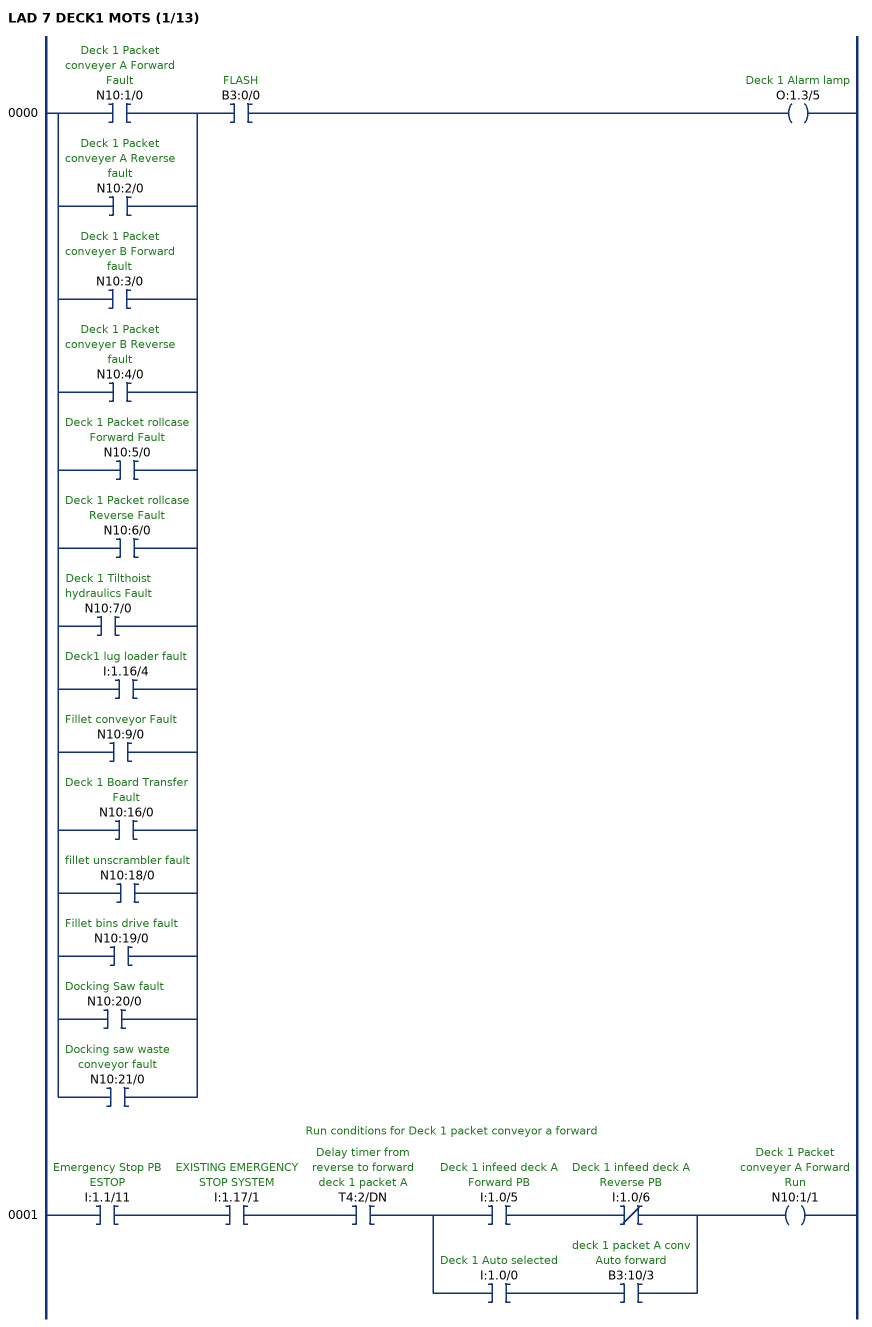
% Rung: 0 %
SOR BST XIC N10:1/0 NXB XIC N10:2/0 NXB XIC N10:3/0 NXB XIC N10:4/0 NXB XIC N10:5/0 NXB XIC N10:6/0 NXB XIC N10:7/0 NXB XIC I:1.16/4 NXB XIC N10:9/0 NXB XIC N10:16/0 NXB XIC N10:18/0 NXB XIC N10:19/0 NXB XIC N10:20/0 NXB XIC N10:21/0 BND XIC B3:0/0 OTE O:1.3/5 EOR
%   N10:1/0  "Deck 1 Packet conveyer A Forward Fault" %
%   N10:2/0  "Deck 1 Packet conveyer A Reverse fault" %
%   N10:3/0  "Deck 1 Packet conveyer B Forward fault" %
%   N10:4/0  "Deck 1 Packet conveyer B Reverse fault" %
%   N10:5/0  "Deck 1 Packet rollcase Forward Fault" %
%   N10:6/0  "Deck 1 Packet rollcase Reverse Fault" %
%   N10:7/0  "Deck 1 Tilthoist hydraulics Fault" %
%   I:1.16/4  "Deck1 lug loader fault" %
%   N10:9/0  "Fillet conveyor Fault" %
%   N10:16/0  "Deck 1 Board Transfer Fault" %
%   N10:18/0  "fillet unscrambler fault" %
%   N10:19/0  "Fillet bins drive fault" %
%   N10:20/0  "Docking Saw fault" %
%   N10:21/0  "Docking saw waste conveyor fault" %
%   B3:0/0  FLASH %
%   O:1.3/5  "Deck 1 Alarm lamp" %
% Rung: 1 %
% Run conditions for Deck 1 packet conveyor a forward %
SOR XIC I:1.1/11 XIC I:1.17/1 XIC T4:2/DN BST XIC I:1.0/5 XIO I:1.0/6 NXB XIC I:1.0/0 XIC B3:10/3 BND OTE N10:1/1 EOR
%   I:1.1/11  ESTOP  "Emergency Stop PB" %
%   I:1.17/1  "EXISTING EMERGENCY STOP SYSTEM" %
%   T4:2/DN  "Delay timer from reverse to forward deck 1 packet A" %
%   I:1.0/5  "Deck 1 infeed deck A Forward PB" %
%   I:1.0/6  "Deck 1 infeed deck A Reverse PB" %
%   I:1.0/0  "Deck 1 Auto selected" %
%   B3:10/3  "deck 1 packet A conv Auto forward" %
%   N10:1/1  "Deck 1 Packet conveyer A Forward Run" %

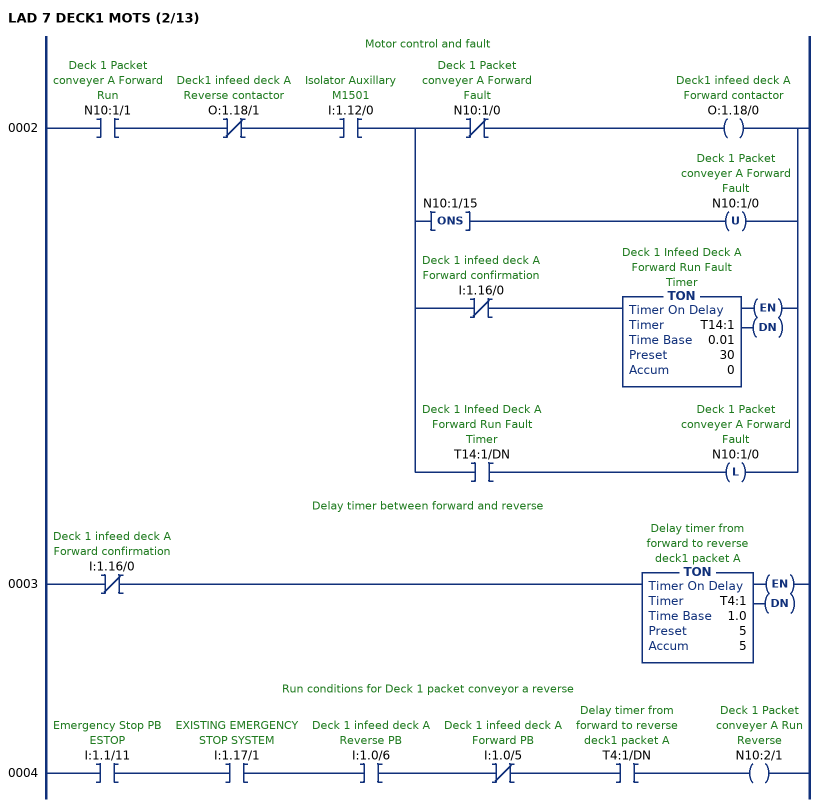
% Rung: 2 %
% Motor control and fault %
SOR XIC N10:1/1 XIO O:1.18/1 XIC I:1.12/0 BST XIO N10:1/0 OTE O:1.18/0 NXB OSR N10:1/15 OTU N10:1/0 NXB XIO I:1.16/0 TON T14:1 0.01 30 0 NXB XIC T14:1/DN OTL N10:1/0 BND EOR
%   N10:1/1  "Deck 1 Packet conveyer A Forward Run" %
%   O:1.18/1  "Deck1 infeed deck A Reverse contactor" %
%   I:1.12/0  "Isolator Auxillary M1501" %
%   N10:1/0  "Deck 1 Packet conveyer A Forward Fault" %
%   O:1.18/0  "Deck1 infeed deck A Forward contactor" %
%   I:1.16/0  "Deck 1 infeed deck A Forward confirmation" %
%   T14:1  "Deck 1 Infeed Deck A Forward Run Fault Timer" %
% Rung: 3 %
% Delay timer between forward and reverse %
SOR XIO I:1.16/0 TON T4:1 1.0 5 5 EOR
%   I:1.16/0  "Deck 1 infeed deck A Forward confirmation" %
%   T4:1  "Delay timer from forward to reverse deck1 packet A" %
% Rung: 4 %
% Run conditions for Deck 1 packet conveyor a reverse %
SOR XIC I:1.1/11 XIC I:1.17/1 XIC I:1.0/6 XIO I:1.0/5 XIC T4:1/DN OTE N10:2/1 EOR
%   I:1.1/11  ESTOP  "Emergency Stop PB" %
%   I:1.17/1  "EXISTING EMERGENCY STOP SYSTEM" %
%   I:1.0/6  "Deck 1 infeed deck A Reverse PB" %
%   I:1.0/5  "Deck 1 infeed deck A Forward PB" %
%   T4:1/DN  "Delay timer from forward to reverse deck1 packet A" %
%   N10:2/1  "Deck 1 Packet conveyer A Run Reverse" %

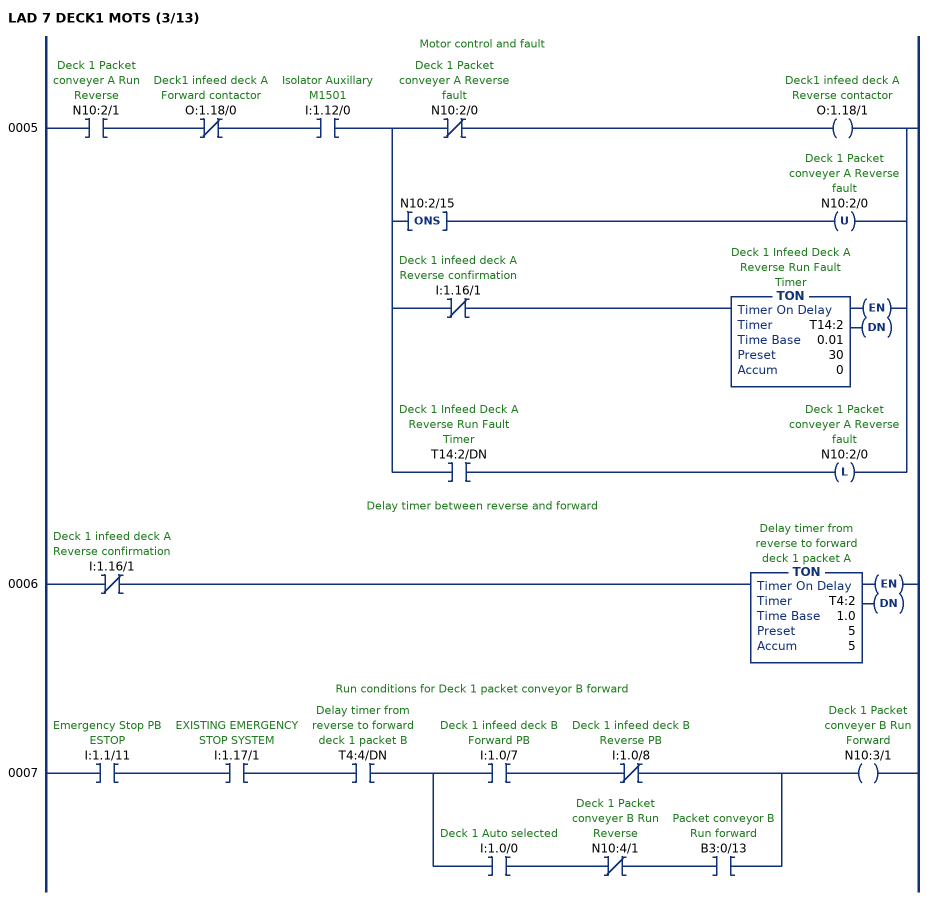
% Rung: 5 %
% Motor control and fault %
SOR XIC N10:2/1 XIO O:1.18/0 XIC I:1.12/0 BST XIO N10:2/0 OTE O:1.18/1 NXB OSR N10:2/15 OTU N10:2/0 NXB XIO I:1.16/1 TON T14:2 0.01 30 0 NXB XIC T14:2/DN OTL N10:2/0 BND EOR
%   N10:2/1  "Deck 1 Packet conveyer A Run Reverse" %
%   O:1.18/0  "Deck1 infeed deck A Forward contactor" %
%   I:1.12/0  "Isolator Auxillary M1501" %
%   N10:2/0  "Deck 1 Packet conveyer A Reverse fault" %
%   O:1.18/1  "Deck1 infeed deck A Reverse contactor" %
%   I:1.16/1  "Deck 1 infeed deck A Reverse confirmation" %
%   T14:2  "Deck 1 Infeed Deck A Reverse Run Fault Timer" %
% Rung: 6 %
% Delay timer between reverse and forward %
SOR XIO I:1.16/1 TON T4:2 1.0 5 5 EOR
%   I:1.16/1  "Deck 1 infeed deck A Reverse confirmation" %
%   T4:2  "Delay timer from reverse to forward deck 1 packet A" %
% Rung: 7 %
% Run conditions for Deck 1 packet conveyor B forward %
SOR XIC I:1.1/11 XIC I:1.17/1 XIC T4:4/DN BST XIC I:1.0/7 XIO I:1.0/8 NXB XIC I:1.0/0 XIO N10:4/1 XIC B3:0/13 BND OTE N10:3/1 EOR
%   I:1.1/11  ESTOP  "Emergency Stop PB" %
%   I:1.17/1  "EXISTING EMERGENCY STOP SYSTEM" %
%   T4:4/DN  "Delay timer from reverse to forward deck 1 packet B" %
%   I:1.0/7  "Deck 1 infeed deck B Forward PB" %
%   I:1.0/8  "Deck 1 infeed deck B Reverse PB" %
%   I:1.0/0  "Deck 1 Auto selected" %
%   N10:4/1  "Deck 1 Packet conveyer B Run Reverse" %
%   B3:0/13  "Packet conveyor B Run forward" %
%   N10:3/1  "Deck 1 Packet conveyer B Run Forward" %

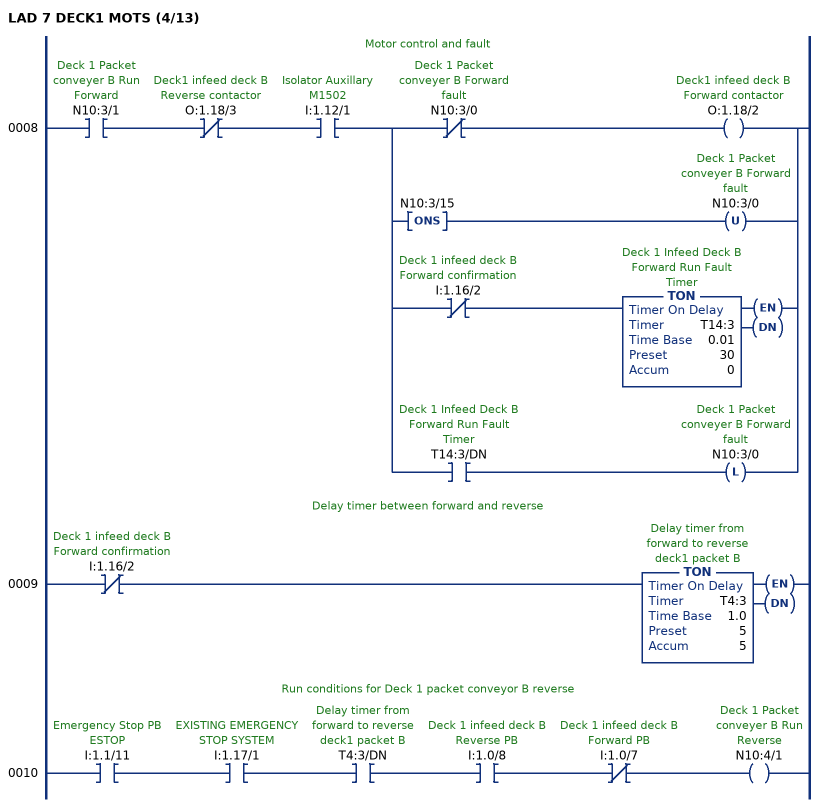
% Rung: 8 %
% Motor control and fault %
SOR XIC N10:3/1 XIO O:1.18/3 XIC I:1.12/1 BST XIO N10:3/0 OTE O:1.18/2 NXB OSR N10:3/15 OTU N10:3/0 NXB XIO I:1.16/2 TON T14:3 0.01 30 0 NXB XIC T14:3/DN OTL N10:3/0 BND EOR
%   N10:3/1  "Deck 1 Packet conveyer B Run Forward" %
%   O:1.18/3  "Deck1 infeed deck B Reverse contactor" %
%   I:1.12/1  "Isolator Auxillary M1502" %
%   N10:3/0  "Deck 1 Packet conveyer B Forward fault" %
%   O:1.18/2  "Deck1 infeed deck B Forward contactor" %
%   I:1.16/2  "Deck 1 infeed deck B Forward confirmation" %
%   T14:3  "Deck 1 Infeed Deck B Forward Run Fault Timer" %
% Rung: 9 %
% Delay timer between forward and reverse %
SOR XIO I:1.16/2 TON T4:3 1.0 5 5 EOR
%   I:1.16/2  "Deck 1 infeed deck B Forward confirmation" %
%   T4:3  "Delay timer from forward to reverse deck1 packet B" %
% Rung: 10 %
% Run conditions for Deck 1 packet conveyor B reverse %
SOR XIC I:1.1/11 XIC I:1.17/1 XIC T4:3/DN XIC I:1.0/8 XIO I:1.0/7 OTE N10:4/1 EOR
%   I:1.1/11  ESTOP  "Emergency Stop PB" %
%   I:1.17/1  "EXISTING EMERGENCY STOP SYSTEM" %
%   T4:3/DN  "Delay timer from forward to reverse deck1 packet B" %
%   I:1.0/8  "Deck 1 infeed deck B Reverse PB" %
%   I:1.0/7  "Deck 1 infeed deck B Forward PB" %
%   N10:4/1  "Deck 1 Packet conveyer B Run Reverse" %

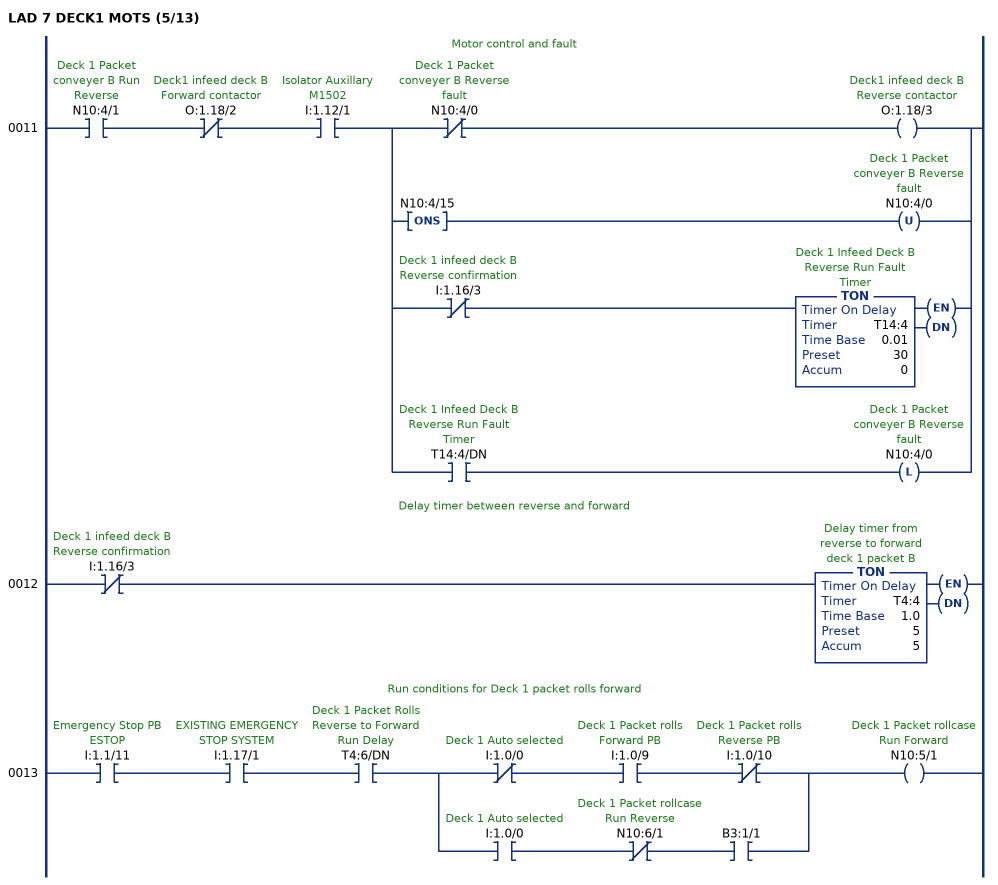
% Rung: 11 %
% Motor control and fault %
SOR XIC N10:4/1 XIO O:1.18/2 XIC I:1.12/1 BST XIO N10:4/0 OTE O:1.18/3 NXB OSR N10:4/15 OTU N10:4/0 NXB XIO I:1.16/3 TON T14:4 0.01 30 0 NXB XIC T14:4/DN OTL N10:4/0 BND EOR
%   N10:4/1  "Deck 1 Packet conveyer B Run Reverse" %
%   O:1.18/2  "Deck1 infeed deck B Forward contactor" %
%   I:1.12/1  "Isolator Auxillary M1502" %
%   N10:4/0  "Deck 1 Packet conveyer B Reverse fault" %
%   O:1.18/3  "Deck1 infeed deck B Reverse contactor" %
%   I:1.16/3  "Deck 1 infeed deck B Reverse confirmation" %
%   T14:4  "Deck 1 Infeed Deck B Reverse Run Fault Timer" %
% Rung: 12 %
% Delay timer between reverse and forward %
SOR XIO I:1.16/3 TON T4:4 1.0 5 5 EOR
%   I:1.16/3  "Deck 1 infeed deck B Reverse confirmation" %
%   T4:4  "Delay timer from reverse to forward deck 1 packet B" %
% Rung: 13 %
% Run conditions for Deck 1 packet rolls forward %
SOR XIC I:1.1/11 XIC I:1.17/1 XIC T4:6/DN BST XIO I:1.0/0 XIC I:1.0/9 XIO I:1.0/10 NXB XIC I:1.0/0 XIO N10:6/1 XIC B3:1/1 BND OTE N10:5/1 EOR
%   I:1.1/11  ESTOP  "Emergency Stop PB" %
%   I:1.17/1  "EXISTING EMERGENCY STOP SYSTEM" %
%   T4:6  "Deck 1 Packet Rolls Reverse to Forward Run Delay" %
%   I:1.0/0  "Deck 1 Auto selected" %
%   I:1.0/9  "Deck 1 Packet rolls Forward PB" %
%   I:1.0/10  "Deck 1 Packet rolls Reverse PB" %
%   N10:6/1  "Deck 1 Packet rollcase Run Reverse" %
%   N10:5/1  "Deck 1 Packet rollcase Run Forward" %

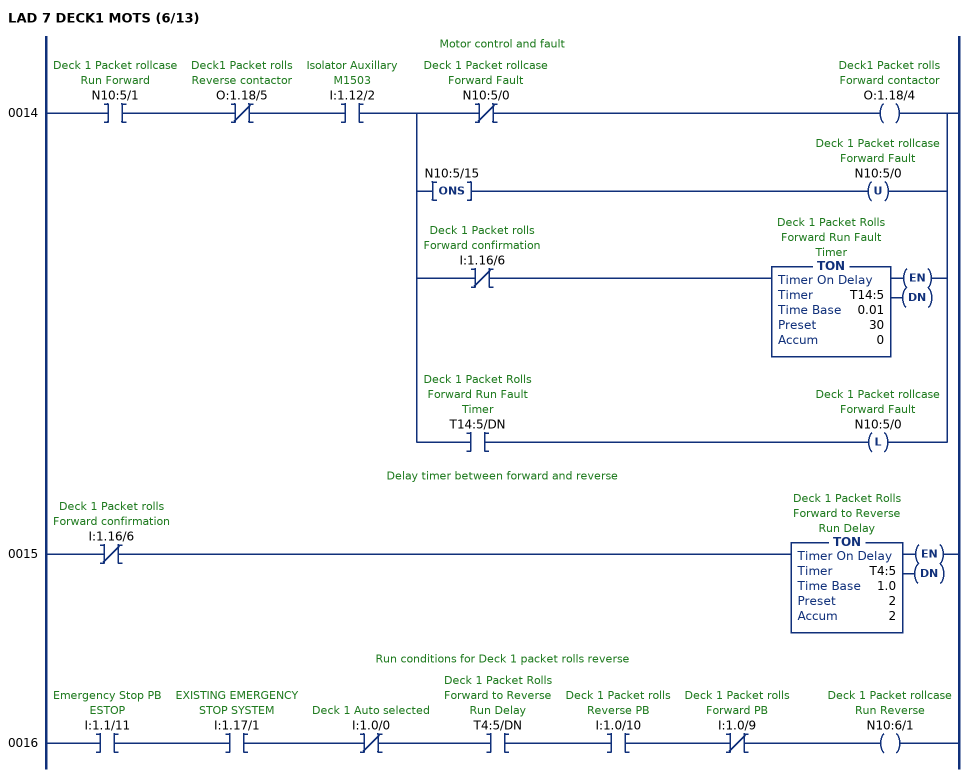
% Rung: 14 %
% Motor control and fault %
SOR XIC N10:5/1 XIO O:1.18/5 XIC I:1.12/2 BST XIO N10:5/0 OTE O:1.18/4 NXB OSR N10:5/15 OTU N10:5/0 NXB XIO I:1.16/6 TON T14:5 0.01 30 0 NXB XIC T14:5/DN OTL N10:5/0 BND EOR
%   N10:5/1  "Deck 1 Packet rollcase Run Forward" %
%   O:1.18/5  "Deck1 Packet rolls Reverse contactor" %
%   I:1.12/2  "Isolator Auxillary M1503" %
%   N10:5/0  "Deck 1 Packet rollcase Forward Fault" %
%   O:1.18/4  "Deck1 Packet rolls Forward contactor" %
%   I:1.16/6  "Deck 1 Packet rolls Forward confirmation" %
%   T14:5  "Deck 1 Packet Rolls Forward Run Fault Timer" %
% Rung: 15 %
% Delay timer between forward and reverse %
SOR XIO I:1.16/6 TON T4:5 1.0 2 2 EOR
%   I:1.16/6  "Deck 1 Packet rolls Forward confirmation" %
%   T4:5  "Deck 1 Packet Rolls Forward to Reverse Run Delay" %
% Rung: 16 %
% Run conditions for Deck 1 packet rolls reverse %
SOR XIC I:1.1/11 XIC I:1.17/1 XIO I:1.0/0 XIC T4:5/DN XIC I:1.0/10 XIO I:1.0/9 OTE N10:6/1 EOR
%   I:1.1/11  ESTOP  "Emergency Stop PB" %
%   I:1.17/1  "EXISTING EMERGENCY STOP SYSTEM" %
%   I:1.0/0  "Deck 1 Auto selected" %
%   T4:5  "Deck 1 Packet Rolls Forward to Reverse Run Delay" %
%   I:1.0/10  "Deck 1 Packet rolls Reverse PB" %
%   I:1.0/9  "Deck 1 Packet rolls Forward PB" %
%   N10:6/1  "Deck 1 Packet rollcase Run Reverse" %

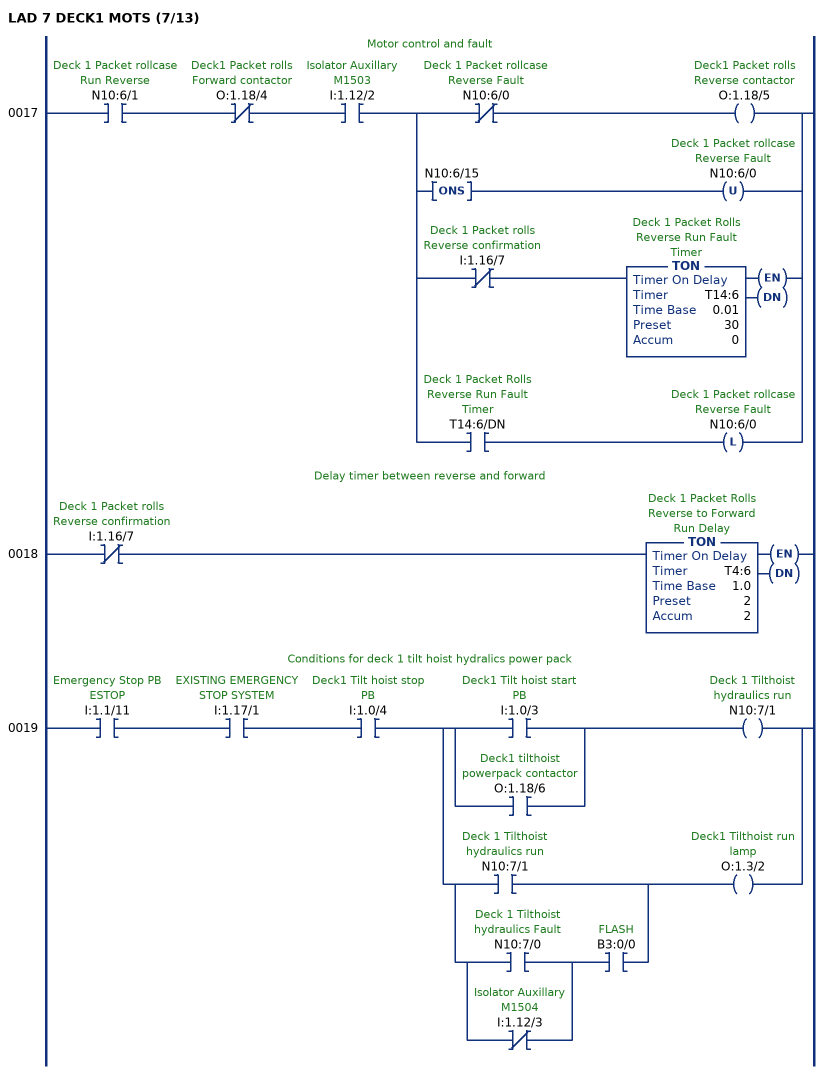
% Rung: 17 %
% Motor control and fault %
SOR XIC N10:6/1 XIO O:1.18/4 XIC I:1.12/2 BST XIO N10:6/0 OTE O:1.18/5 NXB OSR N10:6/15 OTU N10:6/0 NXB XIO I:1.16/7 TON T14:6 0.01 30 0 NXB XIC T14:6/DN OTL N10:6/0 BND EOR
%   N10:6/1  "Deck 1 Packet rollcase Run Reverse" %
%   O:1.18/4  "Deck1 Packet rolls Forward contactor" %
%   I:1.12/2  "Isolator Auxillary M1503" %
%   N10:6/0  "Deck 1 Packet rollcase Reverse Fault" %
%   O:1.18/5  "Deck1 Packet rolls Reverse contactor" %
%   I:1.16/7  "Deck 1 Packet rolls Reverse confirmation" %
%   T14:6  "Deck 1 Packet Rolls Reverse Run Fault Timer" %
% Rung: 18 %
% Delay timer between reverse and forward %
SOR XIO I:1.16/7 TON T4:6 1.0 2 2 EOR
%   I:1.16/7  "Deck 1 Packet rolls Reverse confirmation" %
%   T4:6  "Deck 1 Packet Rolls Reverse to Forward Run Delay" %
% Rung: 19 %
% Conditions for deck 1 tilt hoist hydralics power pack %
SOR XIC I:1.1/11 XIC I:1.17/1 XIC I:1.0/4 BST BST XIC I:1.0/3 NXB XIC O:1.18/6 BND OTE N10:7/1 NXB BST XIC N10:7/1 NXB BST XIC N10:7/0 NXB XIO I:1.12/3 BND XIC B3:0/0 BND OTE O:1.3/2 BND EOR
%   I:1.1/11  ESTOP  "Emergency Stop PB" %
%   I:1.17/1  "EXISTING EMERGENCY STOP SYSTEM" %
%   I:1.0/4  "Deck1 Tilt hoist stop PB" %
%   I:1.0/3  "Deck1 Tilt hoist start PB" %
%   O:1.18/6  "Deck1 tilthoist powerpack contactor" %
%   N10:7/1  "Deck 1 Tilthoist hydraulics run" %
%   N10:7/0  "Deck 1 Tilthoist hydraulics Fault" %
%   I:1.12/3  "Isolator Auxillary M1504" %
%   B3:0/0  FLASH %
%   O:1.3/2  "Deck1 Tilthoist run lamp" %

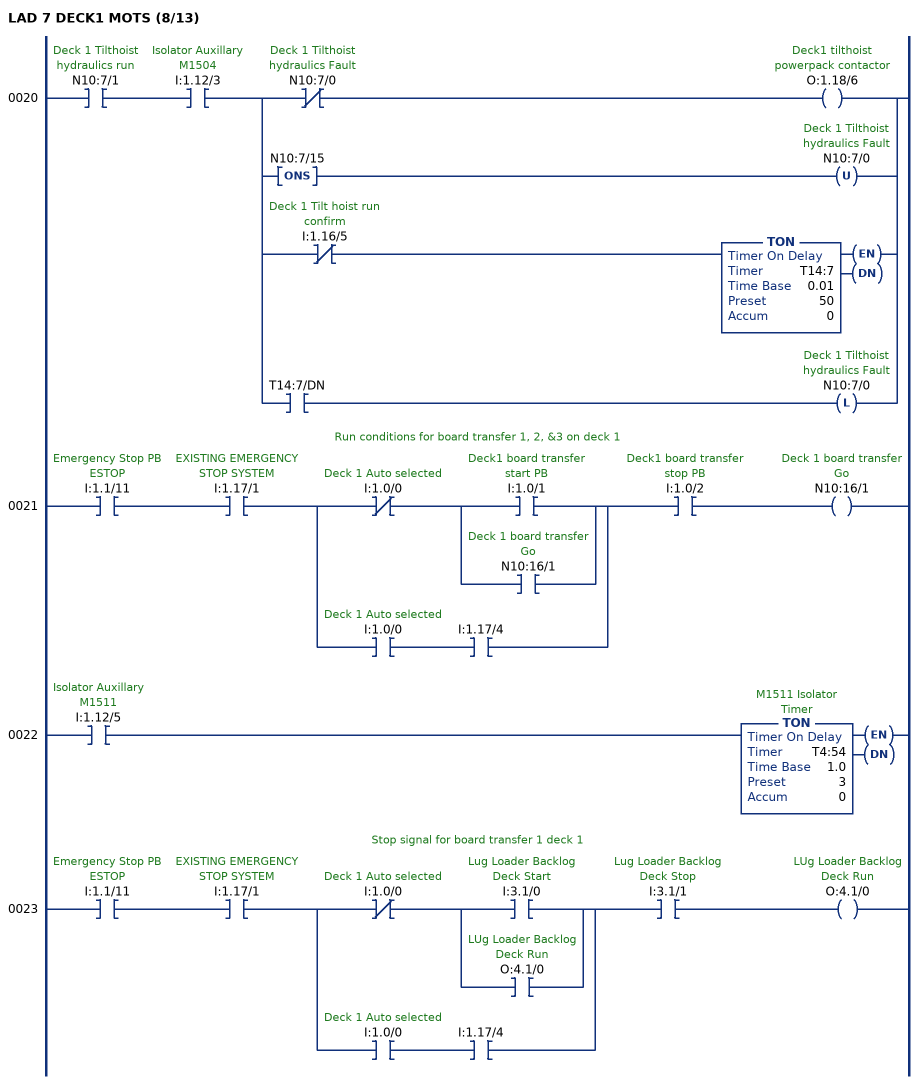
% Rung: 20 %
SOR XIC N10:7/1 XIC I:1.12/3 BST XIO N10:7/0 OTE O:1.18/6 NXB OSR N10:7/15 OTU N10:7/0 NXB XIO I:1.16/5 TON T14:7 0.01 50 0 NXB XIC T14:7/DN OTL N10:7/0 BND EOR
%   N10:7/1  "Deck 1 Tilthoist hydraulics run" %
%   I:1.12/3  "Isolator Auxillary M1504" %
%   N10:7/0  "Deck 1 Tilthoist hydraulics Fault" %
%   O:1.18/6  "Deck1 tilthoist powerpack contactor" %
%   I:1.16/5  "Deck 1 Tilt hoist run confirm" %
% Rung: 21 %
% Run conditions for board transfer 1, 2, &3 on deck 1 %
SOR XIC I:1.1/11 XIC I:1.17/1 BST XIO I:1.0/0 BST XIC I:1.0/1 NXB XIC N10:16/1 BND NXB XIC I:1.0/0 XIC I:1.17/4 BND XIC I:1.0/2 OTE N10:16/1 EOR
%   I:1.1/11  ESTOP  "Emergency Stop PB" %
%   I:1.17/1  "EXISTING EMERGENCY STOP SYSTEM" %
%   I:1.0/0  "Deck 1 Auto selected" %
%   I:1.0/1  "Deck1 board transfer start PB" %
%   N10:16/1  "Deck 1 board transfer Go" %
%   I:1.0/2  "Deck1 board transfer stop PB" %
% Rung: 22 %
SOR XIC I:1.12/5 TON T4:54 1.0 3 0 EOR
%   I:1.12/5  "Isolator Auxillary M1511" %
%   T4:54  "M1511 Isolator Timer" %
% Rung: 23 %
% Stop signal for board transfer 1 deck 1 %
SOR XIC I:1.1/11 XIC I:1.17/1 BST XIO I:1.0/0 BST XIC I:3.1/0 NXB XIC O:4.1/0 BND NXB XIC I:1.0/0 XIC I:1.17/4 BND XIC I:3.1/1 OTE O:4.1/0 EOR
%   I:1.1/11  ESTOP  "Emergency Stop PB" %
%   I:1.17/1  "EXISTING EMERGENCY STOP SYSTEM" %
%   I:1.0/0  "Deck 1 Auto selected" %
%   I:3.1/0  "Lug Loader Backlog Deck Start" %
%   O:4.1/0  "LUg Loader Backlog Deck Run" %
%   I:3.1/1  "Lug Loader Backlog Deck Stop" %

